FUNCTION_BLOCK FB_observerCsv IMPLEMENTS InterfaceObserver
VAR_INPUT
END_VAR
VAR_OUTPUT
	{attribute 'TcEncoding':='UTF-8'}
	text : T_MAXSTRING;
END_VAR
VAR
END_VAR

METHOD subscribe_job_directory : BOOL
VAR_INPUT
	executor	: REFERENCE TO FB_Executor;
END_VAR
VAR
	job_log : STRING;
END_VAR
IF __ISVALIDREF(executor) THEN

	job_log := CONCAT(job_log, 'JOB STRUCTURE');
	IF executor.future <> 0 THEN
		job_log := CONCAT(job_log, '/ FUTURE_NAME : ');
		job_log := CONCAT(job_log, executor.future.future_name);
		job_log := CONCAT(job_log, ', ');	
	END_IF
	job_log := CONCAT(job_log, 'JOB_ID : ');
	job_log := CONCAT(job_log, executor.uid);

	ADSLOGSTR(msgCtrlMask := ADSLOG_MSGTYPE_LOG, msgFmtStr := job_log, strArg := '');
END_IF
END_METHOD

METHOD subscribe_job_event : BOOL
VAR_INPUT
	subject		: T_MaxString;
	old_state	: E_FutureExecutionState;
	new_state	: E_FutureExecutionState;
	record_time	: Tc2_Utilities.T_FILETIME64;
	executor	: REFERENCE TO FB_Executor;
END_VAR
VAR_INST
	fb_timezone_info : FB_GetTimeZoneInformation := (bExecute := TRUE);
END_VAR
VAR
	last_state : STRING;
	current_state : STRING;
	container : InterfaceContainer;
	num_of_jobs : UINT;
END_VAR
last_state := TO_STRING(old_state);
current_state := TO_STRING(new_state);

IF __QUERYINTERFACE(executor.future, container) THEN
	num_of_jobs := container.num_of_jobs;
ELSE
	num_of_jobs := 1;
END_IF


IF __ISVALIDREF(executor) THEN
	fb_timezone_info();
	text := FILETIME64_TO_ISO8601(fileTime := record_time, nBias := DINT_TO_INT(fb_timezone_info.tzInfo.bias), bUTC := TRUE,nPrecision := 6);
	text := CONCAT(text, ',');
	text := CONCAT(text, subject);
	text := CONCAT(text, ',');
	text := CONCAT(text, TO_STRING(current_state));
	text := CONCAT(text, ',');
	text := CONCAT(text, TO_STRING(executor.nErrorID));
	text := CONCAT(text, ',');
	text := CONCAT(text, executor.future.future_name);
	text := CONCAT(text, ',');
	text := CONCAT(text, executor.uid);
	text := CONCAT(text, ',');
	text := CONCAT(text, TO_STRING(num_of_jobs));
	
	
	ADSLOGSTR(msgCtrlMask := ADSLOG_MSGTYPE_LOG,
 			 msgFmtStr := text, 
			strArg := '');	
END_IF

subscribe_job_event := TRUE;
END_METHOD

END_FUNCTION_BLOCK

(* stored: Version 1.1.0.1, ProductVersion 3.1.4024.15
   POU FB_observerCsv: Id {1233ff4c-0021-4e11-b8c0-930aad80ce81}, SpecialFunc None
   Method subscribe_job_directory: Id {6dfb0292-67d2-492c-b8b0-02321a10a38b}
   Method subscribe_job_event: Id {f1619f42-b89d-4ee0-922a-89150dc1d881} *)
